Staubli VAL3: putEx.pgx

public program putEx(num nX, num nY, string sText)
begin
  // Displays a text at the cursor position (x,y)
  //
  // The cursor is positioned on the character after the last character of
  // the message displayed
  //
  // copyright (c) 2015-2018 victortorreslopez
  //
  // GNU General Public License
  //
  // Parameters
  // - nX: cursor column (0 to 39)
  // - nY: cursor row (0 to 13)
  // - sText: character string type expression
  //
  // Version history
  // ---------------
  // 2.0, 2020/02/15, VTL: renames all parameters
  // 1.0, 2018/09/28, VTL: renames "sText" by "s"
  // 0.0, 2015/01/15, VTL: alfa release

  gotoxy(nX, nY)
  put(sText)
end
